Staubli VAL3: Deb2403.pjx

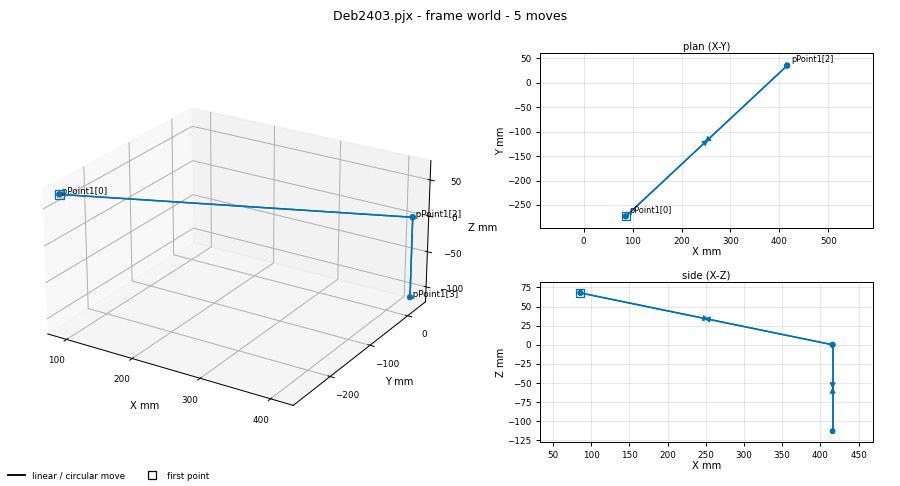
[picture p0: tool path of Deb2403.pjx in frame world, 5 of 9 moves have a stored position in this frame; points joined in program order, loops and branches not executed]
--- Deb2403.pjx ---
Parameters version=s7.4 stackSize=5000 millimeterUnit=true
Program file=main.pgx
Program file=prgm1.pgx
Program file=start.pgx
Program file=stop.pgx
Program file=test_com.pgx
Data file=Deb2403.dtx

--- Deb2403.dtx ---
mdesc mNomSpeed[2]
  [0] = {blend=cartesian}
  [1] = {accel=50, vel=50, decel=50, blend=cartesian}
tool tTool = {z=67, fatherId=flange[0], ioLink=valve1}
jointRx jP1
jointRx jP2 = {j1=67.72, j2=50.87, j3=100.24, j5=28.89, j6=-112.28}
jointRx jP3 = {j1=-83.94, j2=66.93, j3=62.59, j5=50.48, j6=-263.94}
jointRx jP4 = {j1=67.72, j2=17.89, j3=90, j5=72.11, j6=-112.28}
jointRx jP5 = {j1=-84.94, j2=43.97, j3=50.35, j5=58.68, j6=-263.94}
frame fFrame = {x=-421.67, y=-92.07, z=-232.31, rx=0.62, ry=178.2, rz=-83.18, fatherId=world[0]}
public dio diECAT1_0 = {link=POWERLINK-1\%I0}
public dio diECAT1_1 = {link=POWERLINK-1\%I1}
public dio diECAT1_2 = {link=POWERLINK-1\%I2}
public dio diECAT1_3 = {link=POWERLINK-1\%I3}
public dio diECAT1_4 = {link=POWERLINK-1\%I4}
public dio diECAT1_5 = {link=POWERLINK-1\%I5}
public dio diECAT1_6 = {link=POWERLINK-1\%I6}
public dio diECAT1_7 = {link=POWERLINK-1\%I7}
public dio diECAT1_8 = {link=POWERLINK-1\%I8}
public dio diECAT1_9 = {link=POWERLINK-1\%I9}
public dio diECAT1_10 = {link=POWERLINK-1\%I10}
public dio diECAT1_11 = {link=POWERLINK-1\%I11}
public dio diECAT1_12 = {link=POWERLINK-1\%I12}
public dio diECAT1_13 = {link=POWERLINK-1\%I13}
public dio diECAT1_14 = {link=POWERLINK-1\%I14}
public dio diECAT1_15 = {link=POWERLINK-1\%I15}
public dio diECAT1_16 = {link=POWERLINK-1\%I16}
public dio doECAT1_0 = {link=POWERLINK-1\%Q0}
public dio doECAT1_1 = {link=POWERLINK-1\%Q1}
bool rbt_ready
num co_x
num co_y
num nPowerlink
num y[8]
num x[8]
pointRx pPointRx = {x=-203.1, y=-91.7, z=-202.86, ry=180, rz=-87.6, fatherId=world[0]}
trsf trTrsf
pointRx pPoint1[4]
  [0] = {x=86.09, y=-273.22, z=67.88, rx=180, fatherId=world[0]}
  [1] = {x=261.8, y=34.46, z=106.21, rx=180, fatherId=world[0]}
  [2] = {x=415.89, y=34.86, z=0.1, rx=180, fatherId=world[0]}
  [3] = {x=415.89, y=34.97, z=-112.94, rx=180, fatherId=world[0]}
dio valve = {link=valve1}

--- main.pgx ---
program main()
begin
  while true
    doECAT1_0 = true

    if(diECAT1_0 == true)

      doECAT1_0 = false

      if(diECAT1_1 == true)
        x[0] = 1
      else
        x[0] = 0
      endIf
      if(diECAT1_2 == true)
        x[1] = 1
      else
        x[1] = 0
      endIf
      if(diECAT1_3 == true)
        x[2] = 1
      else
        x[2] = 0
      endIf
      if(diECAT1_4 == true)
        x[3] = 1
      else
        x[3] = 0
      endIf
      if(diECAT1_5 == true)
        x[4] = 1
      else
        x[4] = 0
      endIf
      if(diECAT1_6 == true)
        x[5] = 1
      else
        x[5] = 0
      endIf
      if(diECAT1_7 == true)
        x[6] = 1
      else
        x[6] = 0
      endIf
      if(diECAT1_8 == true)
        x[7] = 1
      else
        x[7] = 0
      endIf

      co_x =  (x[0] * 1 + x[1] * 2 + x[2] * 4 + x[3] * 8 + x[4] * 16 + x[5] * 32 + x[6] * 64 + x[7] * 128)

      if(diECAT1_9 == true)
        y[0] = 1
      else
        y[0] = 0
      endIf
      if(diECAT1_10 == true)
        y[1] = 1
      else
        y[1] = 0
      endIf
      if(diECAT1_11 == true)
        y[2] = 1
      else
        y[2] = 0
      endIf
      if(diECAT1_12 == true)
        y[3] = 1
      else
        y[3] = 0
      endIf
      if(diECAT1_13 == true)
        y[4] = 1
      else
        y[4] = 0
      endIf
      if(diECAT1_14 == true)
        y[5] = 1
      else
        y[5] = 0
      endIf
      if(diECAT1_15 == true)
        y[6] = 1
      else
        y[6] = 0
      endIf
      if(diECAT1_16 == true)
        y[7] = 1
      else
        y[7] = 0
      endIf

      co_y = (y[0] * 1 + y[1] * 2 + y[2] * 4 + y[3] * 8 + y[4] * 16 + y[5] * 32 + y[6] * 64 + y[7] * 128)


      movel(appro(pPointRx,{co_x,co_y,0,0,0,0}), tTool, mNomSpeed[1])
      movel(appro(pPointRx,{co_x,co_y,25.46,0,0,0}), tTool, mNomSpeed[1])
      waitEndMove()
      open(tTool)
      movel(appro(pPointRx,{co_x,co_y,0,0,0,0}), tTool, mNomSpeed[0])
      movel(pPoint1[0],tTool,mNomSpeed[0])
      movel(pPoint1[2],tTool,mNomSpeed[1])
      movel(pPoint1[3],tTool,mNomSpeed[1])
      waitEndMove()
      close(tTool)
      movel(pPoint1[2],tTool,mNomSpeed[0])
      movel(pPoint1[0],tTool,mNomSpeed[0])

      doECAT1_0 = true

    endIf
  endWhile
end

--- start.pgx ---
program start()
begin
      call main()
end

--- prgm1.pgx ---
program prgm1()
begin
  co_x = 20
  co_y = -20
  movel(appro(pPointRx,{co_x,co_y,0,0,0,0}), tTool, mNomSpeed)
  waitEndMove()

end
